// TIA Portal V20 export
TYPE "typeUnitCommunicationControlNode"
// stored: Namespace Unit1.Em1
   STRUCT
      BA040 : "Unit1.Em1.typeUnitCommunicationControlNodeBA040";
   END_STRUCT;
END_TYPE
